PROGRAM P_Demo_FB_HVACGetSystemTime
VAR
    fb : FB_HVACGetSystemTime;                            // 被演示 FB 实例
    bEnable_in : BOOL := FALSE;
    sNETID_in : T_AmsNetId ;
    tGetSystemTime_in : TIME := T#0S;
    bGetSystemTime_in : BOOL := FALSE;
    bReadyGetSystemTime_out : BOOL;
    bReadyRTC_out : BOOL;
    stSystemTime_out : TIMESTRUCT;
    dtSystemTime_out : DT;
    uiYear_out : UINT;
    uiMonth_out : UINT;
    uiDay_out : UINT;
    uiDayOfWeek_out : UINT;
    uiHour_out : UINT;
    uiMinute_out : UINT;
    uiSecond_out : UINT;
    uiMilliseconds_out : UINT;
    bErrorGetSystemTime_out : BOOL;
    udiErrorIdGetSystemTime_out : UDINT;
END_VAR

// ============================================================================
// Tc2_HVAC.FB_HVACGetSystemTime 演示程序
// ============================================================================
// 场景：把本 FB 实例化到一个 PLC 程序里，每周期单次调用；按需要把 VAR_INPUT 与
//       VAR_IN_OUT 接到工程信号；VAR_OUTPUT 写入对应监视变量。
// 价值：使用本 FB 比手写状态机 / 控制算法节省大量代码；与 Tc2_HVAC 体系内其它 FB
//       直接对接，命名 / 持久化 / 模式仲裁等约定一致。具体语义见 FB_HVACGetSystemTime.md 主文档。
// 验证步骤：
//   1. 右键 PLC 项目下 POUs 文件夹 → Add → Existing Item → 选本 .TcPOU 文件
//   2. 引用 Tc2_HVAC（References → Add library）
//   3. 编译 → 登录 → 运行
//   4. 在线写各 *_in 输入信号触发 FB；在线 monitor *_out 引脚观察状态
// ============================================================================

fb(
    bEnable := bEnable_in,
    sNETID := sNETID_in,
    tGetSystemTime := tGetSystemTime_in,
    bGetSystemTime := bGetSystemTime_in,
    bReadyGetSystemTime => bReadyGetSystemTime_out,
    bReadyRTC => bReadyRTC_out,
    stSystemTime => stSystemTime_out,
    dtSystemTime => dtSystemTime_out,
    uiYear => uiYear_out,
    uiMonth => uiMonth_out,
    uiDay => uiDay_out,
    uiDayOfWeek => uiDayOfWeek_out,
    uiHour => uiHour_out,
    uiMinute => uiMinute_out,
    uiSecond => uiSecond_out,
    uiMilliseconds => uiMilliseconds_out,
    bErrorGetSystemTime => bErrorGetSystemTime_out,
    udiErrorIdGetSystemTime => udiErrorIdGetSystemTime_out
);

END_PROGRAM

(* stored: Version 1.1.0.1, ProductVersion 3.1.4024.5
   POU P_Demo_FB_HVACGetSystemTime: Id {79c99c41-c932-5d28-805f-d86f85292bb5}, SpecialFunc None *)
